VAR_GLOBAL CONSTANT
	SS_INITIALIZE: SINT := 0;
	SS_STEP: SINT := 1;
END_VAR

(* stored: Version 1.1.0.1, ProductVersion 3.1.4024.13
   GVL G_ControlInit: Id {c153ce31-f431-4dba-9c4d-609dbd7cb04b} *)
